// TIA Portal project "KonveyorVeRobotluCilalamaSistemi" (V17)

(* hardware
DEVICE "S7-1200 station_1"  S7-1200 Station
   slot 0: "Rack_0"  S7-1200 Rack  Rack  V1.0
   slot 1: "PLC_1"  CPU 1214C DC/DC/DC  6ES7 214-1AG40-0XB0  V4.5
*)

// ===== PLC "PLC_1"  CPU 1214C DC/DC/DC =====

VAR_GLOBAL   // PLC tag table "Default tag table"
   "START" AT %I0.0 : Bool;
   "SENSÖR 1" AT %I0.1 : Bool;
   "Tag_1" AT %M0.1 : Bool;
   "KONVEYOR BANT MOTORU" AT %Q0.0 : Bool;
   "SENSÖR 2" AT %I0.3 : Bool;
   "SENSÖR 4" AT %I0.7 : Bool;
   "Tag_2" AT %M0.2 : Bool;
   "ACİL STOP 2" AT %I0.4 : Bool;
   "KONVEYOR 90 DERECE DÖNDÜRME MOTORU" AT %Q0.1 : Bool;
   "SENSÖR 3" AT %I0.5 : Bool;
   "Tag_3" AT %M0.3 : Bool;
   "ACİL STOP 3" AT %I0.6 : Bool;
   "180 DERECE AYIRICI DUVAR DÖNDÜRME MOTORU" AT %Q0.2 : Bool;
   "ACİL STOP 1" AT %I0.2 : Bool;
END_VAR

ORGANIZATION_BLOCK "Main"   // OB1, LAD, ProgramCycle
TITLE = "Main Program Sweep (Cycle)"
{ S7_Optimized_Access := 'TRUE' }
VERSION : 0.1
   VAR_INPUT
      Initial_Call : Bool;   // Initial call of this OB
      Remanence : Bool;   // =True, if remanent data are available
   END_VAR
   VAR_TEMP   // added for the SCL form of the ladder/FBD networks
      _w1 : Bool;
   END_VAR
BEGIN

REGION Network 1
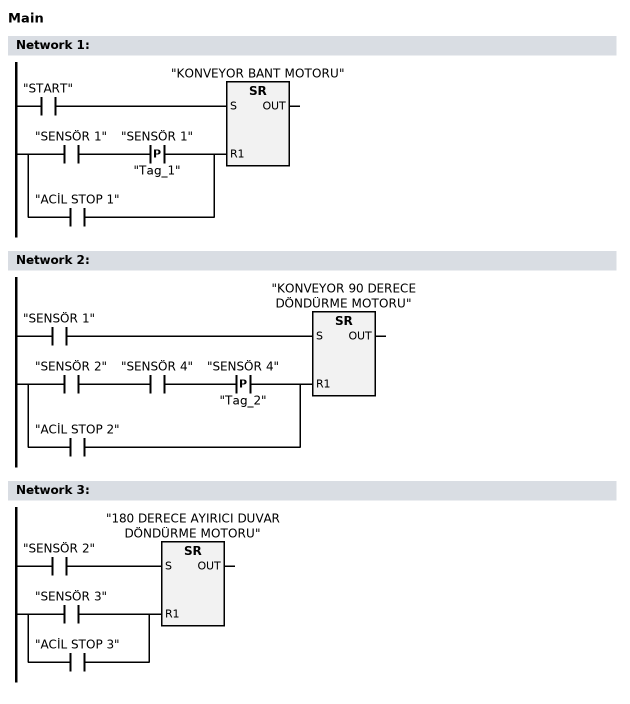
   RUNG wire#powerrail
      Contact( "START" )
      S_SR(operand := "KONVEYOR BANT MOTORU", r1 := wire#w1)
   END_RUNG
   RUNG wire#powerrail
      Contact( "SENSÖR 1" )
      P_Contact(operand := "SENSÖR 1", bit := "Tag_1")
   END_RUNG wire#w1
   RUNG wire#powerrail
      Contact( "ACİL STOP 1" )
   END_RUNG wire#w1
   // the same network as SCL:
   #_w1 := "SENSÖR 1" AND "SENSÖR 1" AND NOT "Tag_1";   // rising edge of "SENSÖR 1"
   "Tag_1" := "SENSÖR 1";
   IF "START" THEN
       "KONVEYOR BANT MOTORU" := TRUE;   // SR flip-flop
   END_IF;
   IF #_w1 OR "ACİL STOP 1" THEN "KONVEYOR BANT MOTORU" := FALSE; END_IF;
END_REGION

REGION Network 2
   RUNG wire#powerrail
      Contact( "SENSÖR 1" )
      S_SR(operand := "KONVEYOR 90 DERECE DÖNDÜRME MOTORU", r1 := wire#w1)
   END_RUNG
   RUNG wire#powerrail
      Contact( "SENSÖR 2" )
      Contact( "SENSÖR 4" )
      P_Contact(operand := "SENSÖR 4", bit := "Tag_2")
   END_RUNG wire#w1
   RUNG wire#powerrail
      Contact( "ACİL STOP 2" )
   END_RUNG wire#w1
   // the same network as SCL:
   #_w1 := "SENSÖR 2" AND "SENSÖR 4" AND "SENSÖR 4" AND NOT "Tag_2";   // rising edge of "SENSÖR 4"
   "Tag_2" := "SENSÖR 4";
   IF "SENSÖR 1" THEN
       "KONVEYOR 90 DERECE DÖNDÜRME MOTORU" := TRUE;   // SR flip-flop
   END_IF;
   IF #_w1 OR "ACİL STOP 2" THEN "KONVEYOR 90 DERECE DÖNDÜRME MOTORU" := FALSE; END_IF;
END_REGION

REGION Network 3
   RUNG wire#powerrail
      Contact( "SENSÖR 2" )
      S_SR(operand := "180 DERECE AYIRICI DUVAR DÖNDÜRME MOTORU", r1 := wire#w1)
   END_RUNG
   RUNG wire#powerrail
      Contact( "SENSÖR 3" )
   END_RUNG wire#w1
   RUNG wire#powerrail
      Contact( "ACİL STOP 3" )
   END_RUNG wire#w1
   // the same network as SCL:
   IF "SENSÖR 2" THEN
       "180 DERECE AYIRICI DUVAR DÖNDÜRME MOTORU" := TRUE;   // SR flip-flop
   END_IF;
   IF "SENSÖR 3" OR "ACİL STOP 3" THEN "180 DERECE AYIRICI DUVAR DÖNDÜRME MOTORU" := FALSE; END_IF;
END_REGION
END_ORGANIZATION_BLOCK